FUNCTION_BLOCK CollisionGroup IMPLEMENTS I_Cyclic, I_CollisionGroup, I_Resettable, I_Object
VAR_INPUT
END_VAR
VAR_OUTPUT
END_VAR
VAR
	stGroupInformation : CAGroupInfo;
	_caGroup : Tc3_McCoordinatedMotion.AXES_GROUP_REF;
	_ICaGroup : I_Mc2CaGroup;
	ReadGroupStatus : Tc3_McCoordinatedMotion.MC_GroupReadStatus;
	resetCAGroup : ResetGroup(THIS^);
	enableCAGroup : EnableGroup(THIS^);
	disableCAGroup : DisableGroup(THIS^);
	addMover : AddMoverToGroupTask(THIS^);
	removeAllAxes : RemoveAllMoverFromGroup(THIS^);
	grpStop : StopMoverGroup(THIS^);
	removeMover : RemoveMoverFromGroup(THIS^);
	_MyName: STRING;
END_VAR

{analysis -2}

METHOD AddMoverToThisGroup : HRESULT
VAR_INPUT
	MoverToAdd : I_XtsMover;
END_VAR
IF NOT addMover.Busy THEN
	addMover.AddMover(MoverToAdd := MoverToAdd);
	MoverToAdd.MyCAGroup  := THIS^;
	AddMoverToThisGroup := 2;
END_IF
END_METHOD

PROPERTY CAGroupXtsIoEnvInterface : I_Mc2CaGroup
GET
CAGroupXtsIoEnvInterface := _ICaGroup;
END_GET
SET
_ICaGroup := CAGroupXtsIoEnvInterface;
_MyName := _ICaGroup.GetObjectName();
END_SET
END_PROPERTY

METHOD Cycle : HRESULT
VAR
	ResetCaGroupResult : HRESULT;
	EnableCaGroupResult : HRESULT;
	DisableCaGroupResult : HRESULT;
	AddMoverCallResult: HRESULT;
	RemoveAllCycleResult: HRESULT;
	GrpStopCycleResult: HRESULT;
END_VAR
IF _ICaGroup <> 0 THEN
	ReadGroupStatus(
	AxesGroup:= _caGroup, 
	Enable:= TRUE );
	ResetCaGroupResult := resetCAGroup.Cycle();
	EnableCaGroupResult := enableCAGroup.Cycle();
	DisableCaGroupResult := disableCAGroup.Cycle();
	AddMoverCallResult := addMover.Cycle();
	RemoveAllCycleResult := removeAllAxes.Cycle();
	GrpStopCycleResult := grpStop.Cycle();
	removeMover.Cycle();
	
	//Cyclic get CaGroup information
	stGroupInformation.sName := 'MainCAGroup';
	stGroupInformation.eGroupState := _caGroup.NcToPlc.Common.GroupStatus.State;
	stGroupInformation.nAxesCount	:= UDINT_TO_INT(_caGroup.NcToPlc.Common.GroupAxesCount);
	stGroupInformation.nId			:= _caGroup.NcToPlc.Common.GroupOID;	
	Cycle := 1;
ELSE
	Cycle := -1;
END_IF
END_METHOD

METHOD Disable : BOOL
VAR_INPUT
END_VAR
IF NOT disableCAGroup.Busy THEN
	disableCAGroup.Execute();
END_IF
END_METHOD

METHOD Enable : BOOL
VAR_INPUT
END_VAR
IF NOT enableCAGroup.Busy THEN
	enableCAGroup.Execute();
END_IF
END_METHOD

METHOD GetAxisCount : udint
VAR_INPUT
END_VAR
GetAxisCount := _caGroup.NcToPlc.Common.GroupAxesCount;
END_METHOD

PROPERTY GroupRef : reference to AXES_GROUP_REF
GET
GroupRef REF= _caGroup;
END_GET
END_PROPERTY

PROPERTY GroupState : CAGroupStatus
GET
IF ReadGroupStatus.GroupDisabled THEN
	GroupState := CAGroupStatus.mcGroupStateDisabled;
ELSIF ReadGroupStatus.GroupErrorStop THEN
	GroupState := CAGroupStatus.mcGroupStateErrorStop;
ELSIF ReadGroupStatus.GroupHoming THEN
	GroupState := CAGroupStatus.mcGroupStateHoming;
ELSIF ReadGroupStatus.GroupMoving THEN
	GroupState := CAGroupStatus.mcGroupStateMoving;
ELSIF ReadGroupStatus.GroupNotReady THEN
	GroupState := CAGroupStatus.mcGroupStateNotReady;
ELSIF ReadGroupStatus.GroupStandby THEN
	GroupState := CAGroupStatus.mcGroupStateStandby;
ELSIF ReadGroupStatus.GroupStopping THEN
	GroupState := CAGroupStatus.mcGroupStateStopping;
ELSIF ReadGroupStatus.Error THEN
	GroupState := CAGroupStatus.mcGroupError;
END_IF
END_GET
END_PROPERTY

METHOD GroupStop : HRESULT
VAR_INPUT
END_VAR
IF NOT grpStop.Busy THEN
	GroupStop := 2;
	grpStop.Execute();
END_IF
END_METHOD

PROPERTY MyName : string
GET
MyName := _MyName;
END_GET
END_PROPERTY

METHOD RegisterWithParent
VAR_INPUT
	Runner	: I_HostObjects;
END_VAR
Runner.RegisterCyclic(THIS^);
END_METHOD

METHOD RemoveAllMovers : HRESULT
VAR_INPUT
END_VAR
IF NOT removeAllAxes.Busy THEN
	removeAllAxes.RemoveAllMover();
	RemoveAllMovers := 2;
END_IF
END_METHOD

METHOD RemoveAMover : BOOL
VAR_INPUT
	moverId : UDINT;
END_VAR
IF NOT removeMover.Busy THEN
	removeMover.Execute(moverid);
END_IF
END_METHOD

METHOD Reset : HRESULT
IF NOT resetCAGroup.Busy THEN
	resetCAGroup.Execute();
END_IF
END_METHOD

END_FUNCTION_BLOCK

(* stored: Version 1.1.0.1
   POU CollisionGroup: Id {8907fd76-d392-4030-a5c6-041188f5b990}, SpecialFunc None
   Folder Commands: Id {8586cf21-15e1-44d9-a164-c4e3c5e15810}
   Folder Status: Id {f0a1ad0e-7de5-4634-834b-41b20fa92032}
   Method AddMoverToThisGroup: Id {9f418b4e-0cf8-4b65-9d2d-7e6c1a46690c}
   Property CAGroupXtsIoEnvInterface: Id {212be6c7-141f-4d0f-8757-6216cdee75b6}
   Get Get: Id {58823424-db7c-4e8e-8355-ea0d3f334737}
   Set Set: Id {4e382846-3fb7-428a-a6d3-609bca8b4701}
   Method Cycle: Id {6b3cc58f-cb00-45fb-b855-5eb19dbaab5d}
   Method Disable: Id {236769ac-ee48-442c-86de-25258567af7c}
   Method Enable: Id {9a19e9ba-2611-4357-a3d4-698f998ad87d}
   Method GetAxisCount: Id {45b9081d-ba05-41c5-b1b6-c67859faca98}
   Property GroupRef: Id {05d388ea-a899-4954-b35a-8298ecb26dd6}
   Get Get: Id {9960c5ab-7079-4a22-9f43-e4d1a1a5992b}
   Property GroupState: Id {a7850ad8-4f08-4a22-bf4c-efbfd8c96cf5}
   Get Get: Id {51b877d1-f5c7-479f-9b28-cdb51e8876b7}
   Method GroupStop: Id {96e619f0-ba68-4e46-ba5e-bd7a0dcefde6}
   Property MyName: Id {e6811d98-40d4-4440-8374-6ce3386e7963}
   Get Get: Id {e4b2e201-13a7-44e4-888f-38c692b30d08}
   Method RegisterWithParent: Id {0f4efa96-221e-4b5f-b62b-0cd9b26287ac}
   Method RemoveAllMovers: Id {72daaa8f-92d0-4f12-b8f9-45742cf249d6}
   Method RemoveAMover: Id {c380af90-39ac-42df-b7a5-a3aab3a831b8}
   Method Reset: Id {109a65fd-df03-46ac-84a7-fd0107d964ee} *)
